(*	HMI variables

	This block holds all HMI variables and handles communication with the HMI
	
	2024-02 HP
		-initial
*)
{attribute 'no_explicit_call' := 'do not call this POU directly'}
FUNCTION_BLOCK HMI_TemplateClean EXTENDS HMI_BaseBlock

//HMI variables that can be written to by the plc and HMI 
VAR_INPUT
	//Do not change these names, the HMI is hardcoded to use these exact names
	MAN:HMI_MAN_TemplateClean;				//HMI manuals
	STS:HMI_STS_TemplateClean;				//HMI statusses
	WRN:HMI_WRN_TemplateClean;				//HMI warnings
	ERR:HMI_ERR_TemplateClean;				//HMI errors
END_VAR

//Hmi variables that can only be written to by the HMI and read by the plc
VAR_OUTPUT PERSISTENT
	//Do not change these names, the HMI is hardcoded to use these exact names
	SP:HMI_SP_TemplateClean;				//HMI setpoints
END_VAR

//this block should not be called

END_FUNCTION_BLOCK

(* stored: Version 1.1.0.1
   POU HMI_TemplateClean: Id {63ea45a1-a2d1-0730-182b-0dbe59611462}, SpecialFunc None *)
